PROGRAM MAIN
VAR
END_VAR

LD_Logic();

END_PROGRAM

(* stored: Version 1.1.0.1, ProductVersion 3.1.4024.12
   POU MAIN: Id {bfa8e972-5c53-4416-bafc-48217ad68b02}, SpecialFunc None *)
